TYPE ST_watertank_Output :
STRUCT
	Out1: LREAL;
END_STRUCT
END_TYPE

(* stored: Version 1.1.0.1, ProductVersion 3.1.4024.4
   DUT ST_watertank_Output: Id {1a2bb09a-9ae6-4cdb-b47f-227165331b39} *)
